{attribute addProperty BoxType "EL1262-0000-0002"}
{attribute addProperty Id "Ch1_InputAT %I*BOOL81"}
{attribute addProperty CRC "4254832157"}
{attribute addProperty SizeInBites "8"}
{attribute addProperty SizeInBytes "1"}
TYPE Ch1_Input_FD9B961D :
STRUCT
	{attribute addProperty Name "Ch1_Input"}
	Ch1_Input AT %I* : BOOL;
END_STRUCT
END_TYPE

(* stored: Version 1.2.0.0, ProductVersion 3.1.4024.9
   DUT Ch1_Input_FD9B961D: Id {1061aa2d-1593-4c6e-b7c3-309bb4123e73} *)
